FUNCTION_BLOCK WP_AND (* Basic Function Block Type *)
  (* Standard: 61499-2 *)
  (* Version 0.0, 2/7/2012, XPMUser, nxtControl GmbH, Template *)
  PACKAGE Main;
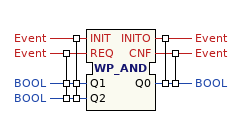
  EVENT_INPUT
    INIT WITH Q1, Q2; (* Initialization Request *)
    REQ WITH Q1, Q2; (* Normal Execution Request *)
  END_EVENT
  EVENT_OUTPUT
    INITO WITH Q0; (* Initialization Confirm *)
    CNF WITH Q0; (* Execution Confirmation *)
  END_EVENT
  VAR_INPUT
    Q1 : BOOL; (* Input event qualifier *)
    Q2 : BOOL;
  END_VAR
  VAR_OUTPUT
    Q0 : BOOL; (* Output event qualifier *)
  END_VAR
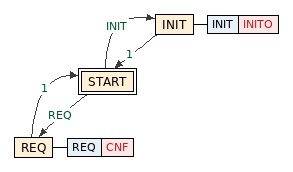
  EC_STATES
    START; (* Initial State *)
    INIT : INIT -> INITO; (* Initialization *)
    REQ : REQ -> CNF; (* Normal execution *)
  END_STATES
  EC_TRANSITIONS
    START TO INIT := INIT;
    INIT TO START := 1;
    START TO REQ := REQ;
    REQ TO START := 1;
  END_TRANSITIONS
  ALGORITHM INIT IN ST: (* Initialization algorithm *)
IF Q1 = TRUE AND Q2 = TRUE THEN
    Q0 := TRUE;
ELSE
    Q0 := FALSE;
END_IF;
  END_ALGORITHM
  ALGORITHM REQ IN ST: (* Normally executed algorithm *)
IF Q1 = TRUE AND Q2 = TRUE THEN
    Q0 := TRUE;
ELSE
    Q0 := FALSE;
END_IF;
  END_ALGORITHM
END_FUNCTION_BLOCK
